{attribute addProperty BoxType "IODEVICETYPE_ETHERCATPROT"}
{attribute addProperty Id "EK1100_Beckhoff_AMI8xxxEK1100_Beckhoff_AMI8xxx_4205BDB361276.5SyncUnitsSyncUnits_CAB22D3B19524.375InputsInputs_C75D3FEC1280160OutputsOutputs_47D1E803848106InfoDataInfoData_E9F65A829612"}
{attribute addProperty CRC "4275013570"}
{attribute addProperty SizeInBites "3031"}
{attribute addProperty SizeInBytes "378.875"}
TYPE EtherCAT_Master_AMIxxxx_FECF87C2 :
STRUCT
	{attribute addProperty Name "EK1100_Beckhoff_AMI8xxx"}
	EK1100_Beckhoff_AMI8xxx : EK1100_Beckhoff_AMI8xxx_4205BDB3;
	{attribute addProperty Name "SyncUnits"}
	SyncUnits : SyncUnits_CAB22D3B;
	{attribute addProperty Name "Inputs"}
	Inputs : Inputs_C75D3FEC;
	{attribute addProperty Name "Outputs"}
	Outputs : Outputs_47D1E803;
	{attribute addProperty Name "InfoData"}
	InfoData : InfoData_E9F65A82;
END_STRUCT
END_TYPE

(* stored: Version 1.2.0.0, ProductVersion 3.1.4024.9
   DUT EtherCAT_Master_AMIxxxx_FECF87C2: Id {c4a1dcc0-feb3-4106-96dd-7d71da5c1bfb} *)
